    aSintDummy22 : ARRAY[0..3] OF SINT := [-128, 127, -34, 104];
    bSintDummy22 : ARRAY[0..3] OF SINT := [-128, 127, -34, 105];

    aSintDummy23 : ARRAY[0..3] OF SINT := [-128, 127, -34, 106];
    bSintDummy23 : ARRAY[0..3] OF SINT := [-128, 127, -34, 107];

    aSintDummy24 : ARRAY[0..3] OF SINT := [-128, 127, -34, 108];
    bSintDummy24 : ARRAY[0..3] OF SINT := [-128, 127, -34, 109];

    aSintDummy25 : ARRAY[0..3] OF SINT := [-128, 127, -34, 110];
    bSintDummy25 : ARRAY[0..3] OF SINT := [-128, 127, -34, 111];

    aSintDummy26 : ARRAY[0..3] OF SINT := [-128, 127, -34, 112];
    bSintDummy26 : ARRAY[0..3] OF SINT := [-128, 127, -34, 113];
END_VAR
TEST('TestWith46FailedArrayAssertions');

AssertArrayEquals_BOOL(Expecteds := aBool,
                       Actuals := bBool,
                       Message := 'Arrays differ');

AssertArrayEquals_BYTE(Expecteds := aByte,
                       Actuals := bByte,
                       Message := 'Arrays differ');

AssertArrayEquals_DINT(Expecteds := aDint,
                       Actuals := bDint,
                       Message := 'Arrays differ');

AssertArrayEquals_DWORD(Expecteds := aDword,
                        Actuals := bDword,
                        Message := 'Arrays differ');

AssertArrayEquals_DWORD(Expecteds := aDword2,
                        Actuals := bDword2,
                        Message := 'Arrays differ');

AssertArrayEquals_INT(Expecteds := aInt,
                      Actuals := bInt,
                      Message := 'Arrays differ');

AssertArrayEquals_LINT(Expecteds := aLint,
                      Actuals := bLint,
                      Message := 'Arrays differ');

AssertArrayEquals_LREAL(Expecteds := aLreal,
                        Actuals := bLreal,
                        Delta := 0.01,
                        Message := 'Arrays differ');

AssertArray2dEquals_LREAL(Expecteds := aLreal2d,
                          Actuals := bLreal2d,
                          Delta := 0.01,
                          Message := 'Arrays differ');

AssertArray3dEquals_LREAL(Expecteds := aLreal3d,
                          Actuals := bLreal3d,
                          Delta := 0.01,
                          Message := 'Arrays differ');

AssertArrayEquals_LWORD(Expecteds := aLword,
                        Actuals := bLword,
                        Message := 'Arrays differ');

AssertArrayEquals_REAL(Expecteds := aReal,
                       Actuals := bReal,
                       Delta := 0.01,
                       Message := 'Arrays differ');

AssertArray2dEquals_REAL(Expecteds := aReal2d,
                         Actuals := bReal2d,
                         Delta := 0.01,
                         Message := 'Arrays differ');

AssertArray3dEquals_REAL(Expecteds := aReal3d,
                         Actuals := bReal3d,
                         Delta := 0.01,
                         Message := 'Arrays differ');

AssertArrayEquals_SINT(Expecteds := aSint,
                       Actuals := bSint,
                       Message := 'Arrays differ');

AssertArrayEquals_UDINT(Expecteds := aUdint,
                        Actuals := bUdint,
                        Message := 'Arrays differ');

AssertArrayEquals_UINT(Expecteds := aUint,
                       Actuals := bUint,
                       Message := 'Arrays differ');

AssertArrayEquals_ULINT(Expecteds := aUlint,
                        Actuals := bUlint,
                        Message := 'Arrays differ');

AssertArrayEquals_USINT(Expecteds := aUsint,
                        Actuals := bUsint,
                        Message := 'Arrays differ');

AssertArrayEquals_WORD(Expecteds := aWord,
                       Actuals := bWord,
                       Message := 'Arrays differ');

AssertArrayEquals_SINT(Expecteds := aSintDummy1,
                       Actuals := bSintDummy1,
                       Message := 'Arrays differ');

AssertArrayEquals_SINT(Expecteds := aSintDummy2,
                       Actuals := bSintDummy2,
                       Message := 'Arrays differ');

AssertArrayEquals_SINT(Expecteds := aSintDummy3,
                       Actuals := bSintDummy3,
                       Message := 'Arrays differ');

AssertArrayEquals_SINT(Expecteds := aSintDummy4,
                       Actuals := bSintDummy4,
                       Message := 'Arrays differ');

AssertArrayEquals_SINT(Expecteds := aSintDummy5,
                       Actuals := bSintDummy5,
                       Message := 'Arrays differ');

AssertArrayEquals_SINT(Expecteds := aSintDummy6,
                       Actuals := bSintDummy6,
                       Message := 'Arrays differ');

AssertArrayEquals_SINT(Expecteds := aSintDummy7,
                       Actuals := bSintDummy7,
                       Message := 'Arrays differ');

AssertArrayEquals_SINT(Expecteds := aSintDummy8,
                       Actuals := bSintDummy8,
                       Message := 'Arrays differ');

AssertArrayEquals_SINT(Expecteds := aSintDummy9,
                       Actuals := bSintDummy9,
                       Message := 'Arrays differ');

AssertArrayEquals_SINT(Expecteds := aSintDummy10,
                       Actuals := bSintDummy10,
                       Message := 'Arrays differ');

AssertArrayEquals_SINT(Expecteds := aSintDummy11,
                       Actuals := bSintDummy11,
                       Message := 'Arrays differ');

AssertArrayEquals_SINT(Expecteds := aSintDummy12,
                       Actuals := bSintDummy12,
                       Message := 'Arrays differ');

AssertArrayEquals_SINT(Expecteds := aSintDummy13,
                       Actuals := bSintDummy13,
                       Message := 'Arrays differ');

AssertArrayEquals_SINT(Expecteds := aSintDummy14,
                       Actuals := bSintDummy14,
                       Message := 'Arrays differ');

AssertArrayEquals_SINT(Expecteds := aSintDummy15,
                       Actuals := bSintDummy15,
                       Message := 'Arrays differ');

AssertArrayEquals_SINT(Expecteds := aSintDummy16,
                       Actuals := bSintDummy16,
                       Message := 'Arrays differ');

AssertArrayEquals_SINT(Expecteds := aSintDummy17,
                       Actuals := bSintDummy17,
                       Message := 'Arrays differ');

AssertArrayEquals_SINT(Expecteds := aSintDummy18,
                       Actuals := bSintDummy18,
                       Message := 'Arrays differ');

AssertArrayEquals_SINT(Expecteds := aSintDummy19,
                       Actuals := bSintDummy19,
                       Message := 'Arrays differ');

AssertArrayEquals_SINT(Expecteds := aSintDummy20,
                       Actuals := bSintDummy20,
                       Message := 'Arrays differ');

AssertArrayEquals_SINT(Expecteds := aSintDummy21,
                       Actuals := bSintDummy21,
                       Message := 'Arrays differ');

AssertArrayEquals_SINT(Expecteds := aSintDummy22,
                       Actuals := bSintDummy22,
                       Message := 'Arrays differ');

AssertArrayEquals_SINT(Expecteds := aSintDummy23,
                       Actuals := bSintDummy23,
                       Message := 'Arrays differ');

AssertArrayEquals_SINT(Expecteds := aSintDummy24,
                       Actuals := bSintDummy1,
                       Message := 'Arrays differ');

AssertArrayEquals_SINT(Expecteds := aSintDummy25,
                       Actuals := bSintDummy1,
                       Message := 'Arrays differ');

AssertArrayEquals_SINT(Expecteds := aSintDummy26,
                       Actuals := bSintDummy26,
                       Message := 'Arrays differ');

TEST_FINISHED();
END_METHOD

END_FUNCTION_BLOCK

// ---- Test/FB_TestDurationMeasurement.TcPOU
(* This testsuite tests that durations are calculated correctly by different types of test cases
    Tests are considered passing if the duration returned is reasonablly close to the expected value.
*)
FUNCTION_BLOCK FB_TestDurationMeasurement EXTENDS TcUnit.FB_TestSuite

TestNamedTest20msDurationMeasuredCorrectly();
TestOrderedTest30msDurationMeasuredCorrectly();
TestRegularTestDurationMeasuredCorrectly();

METHOD PRIVATE TestOrderedTest30msDurationMeasuredCorrectly
VAR_INST
    DelayTimer : TON;
    Counter : DINT;
END_VAR
IF TEST_ORDERED('TestOrderedTest30msDurationMeasuredCorrectly') THEN
    DelayTimer(IN := TRUE, PT := T#30ms);   

    IF delayTimer.Q THEN
        // Write the approximate duration through an assert message for use by the verifier
        AssertEquals_LREAL(0, 0.03, 0, 'Duration');
    
        TEST_FINISHED();
    END_IF
END_IF
END_METHOD

METHOD TestRegularTestDurationMeasuredCorrectly
VAR_INST
    TestExecuted : BOOL;
    TestStartedAt : LWORD;
    TestDuration : LREAL;
    Counter : DINT;
END_VAR
TEST('TestRegularTestDurationMeasuredCorrectly');

IF NOT TestExecuted THEN
    // Introduce a delay and store the time it takes for evaluation by the test
    // use an assert statement as the delay because it takes quite a bit of time
    // double the value to account for the second assert which will print the message
    TestStartedAt := F_GetCpuCounterAs64bit(GVL_TcUnit.GetCpuCounter);
    AssertEquals_LREAL(0, 10, 0, 'Duration for calculation'); 
    TestDuration := LWORD_TO_LREAL(F_GetCpuCounterAs64bit(GVL_TcUnit.GetCpuCounter) - TestStartedAt) * GVL_TcUnit.HundredNanosecondToSecond * 2.0;
    TestExecuted := TRUE;
END_IF

// Write the duration through an assert message for use by the verifier
AssertEquals_LREAL(0, TestDuration, 0, 'Duration');

TEST_FINISHED();
END_METHOD

METHOD TestNamedTest20msDurationMeasuredCorrectly
VAR_INST
    delayTimer : TON;
END_VAR
TEST('TestNamedTest20msDurationMeasuredCorrectly');

delayTimer(IN := TRUE, PT := T#20ms);

IF delayTimer.Q THEN       
    // Write the approximate duration through an assert message for use by the verifier
    AssertEquals_LREAL(0, 0.02, 0, 'Duration');
    
    TEST_FINISHED_NAMED('TestNamedTest20msDurationMeasuredCorrectly');
END_IF
END_METHOD

END_FUNCTION_BLOCK

// ---- Test/FB_TestFileControl.TcPOU
(*
    Contains tests that verify the FileControl function block methods
*)
FUNCTION_BLOCK FB_TestFileControl EXTENDS TcUnit.FB_TestSuite

Test_FileRead();
Test_FileOpen();
Test_FileWrite();
Test_FileClose();
Test_FileDelete();

METHOD Test_FileClose
VAR
    FileControl : TcUnit.FB_FileControl;
    TestFile : STRING := 'Test_FileClose.txt';
    Mode : SysFile.ACCESS_MODE := SysFile.ACCESS_MODE.AM_APPEND_PLUS;
    Actual : SysFile.SysTypes.RTS_IEC_RESULT;
END_VAR
TEST('Test_FileClose');

FileControl.Open(TestFile, Mode);
Actual := FileControl.Close();

AssertEquals_UDINT(Expected := SysDir.CmpErrors.Errors.ERR_OK,
                   Actual := Actual,
                   Message := 'File close failed');

FileControl.Delete(TestFile);

TEST_FINISHED();
END_METHOD

METHOD Test_FileDelete
VAR
    FileControl : TcUnit.FB_FileControl;
    TestFile : STRING := 'Test_FileDelete.txt';
    Mode : SysFile.ACCESS_MODE := SysFile.ACCESS_MODE.AM_APPEND_PLUS;
    Actual : SysFile.SysTypes.RTS_IEC_RESULT;
END_VAR
TEST('Test_FileDelete');

FileControl.Open(TestFile, Mode);
FileControl.Close();
Actual := FileControl.Delete(TestFile);

AssertEquals_UDINT(Expected := Sysdir.CmpErrors.Errors.ERR_OK,
                   Actual := Actual,
                   Message := 'File deletion failed');

TEST_FINISHED();
END_METHOD

METHOD Test_FileOpen
VAR
    FileControl : FB_FileControl;
    TestFile : STRING := 'Test_FileOpen.txt';
    Mode : SysFile.ACCESS_MODE := SysFile.ACCESS_MODE.AM_APPEND_PLUS;
    Actual : SysFile.SysTypes.RTS_IEC_RESULT;
END_VAR
TEST('Test_FileOpen');

FileControl.Open(TestFile, Mode);

AssertEquals_UDINT(Expected := Sysdir.CmpErrors.Errors.ERR_OK,
                   Actual := Actual,
                   Message := 'File open failed');

FileControl.Close();
FileControl.Delete(TestFile);

TEST_FINISHED();
END_METHOD

METHOD Test_FileRead
VAR
    FileControl : FB_FileControl;
    TestFile : STRING := 'Test_FileRead.txt';
    Mode : SysFile.ACCESS_MODE := SysFile.ACCESS_MODE.AM_APPEND_PLUS;
    Result : SysFile.SysTypes.RTS_IEC_RESULT;
    FileSize : SysFile.SysTypes.RTS_IEC_SIZE;
    WriteContents : STRING(64) := '0KflxSh6C%ixPs8ReCPwFuJu)D$p*qfi66iTj&YKMdpq*EGBGiwgAsOs1s(dci';
    ReadContents : STRING(64);
END_VAR
TEST('Test_FileRead');

FileControl.Open(TestFile, Mode);
FileControl.Write(BufferPointer := ADR(WriteContents), Size := SIZEOF(WriteContents));
FileControl.Close();
FileControl.Open(TestFile, FileAccessMode := SysFile.AM_READ);

Result := FileControl.Read(BufferPointer := ADR(ReadContents), SIZEOF(ReadContents), FileSize => FileSize);

AssertEquals_STRING(Expected := WriteContents,
                    Actual := ReadContents,
                    Message := 'File read failed');

FileControl.Close();
FileControl.Delete(TestFile);

TEST_FINISHED();
END_METHOD

METHOD Test_FileWrite
VAR
    FileControl : FB_FileControl;
    Contents : STRING(64) := 'G#NkAM%Muah+nbwAk&8MnQZ9csi*YAoiGkcKzwvsYz5k@yY)aOz&cvQxXQyI6c';
    TestFile : STRING := 'Test_FileWrite.txt';
    Mode : SysFile.ACCESS_MODE := SysFile.ACCESS_MODE.AM_APPEND_PLUS;
    Actual : SysFile.SysTypes.RTS_IEC_RESULT;
END_VAR
TEST('Test_FileWrite');

FileControl.Open(TestFile, Mode);
Actual := FileControl.Write(BufferPointer := ADR(Contents), Size := SIZEOF(Contents));

AssertEquals_UDINT(Expected := SysDir.CmpErrors.Errors.ERR_OK,
                   Actual := Actual,
                   Message := 'File write failed');

FileControl.Close();
FileControl.Delete(TestFile);

TEST_FINISHED();
END_METHOD

END_FUNCTION_BLOCK

// ---- Test/FB_TestXmlControl.TcPOU
// Contains tests that verify the XmlControl function block methods
FUNCTION_BLOCK FB_TestXmlControl EXTENDS TcUnit.FB_TestSuite
VAR
    Buffer: ARRAY[0..TcUnit.GVL_Param_TcUnit.xUnitBufferSize - 1] OF BYTE;
END_VAR

Test_NewTag();
Test_NewTagNested();
Test_NewParameter();
Test_NewComment();
Test_CloseOpenTag();
Test_CloseTag();
Test_NewTagData();

METHOD PRIVATE Setup
// Clear buffer
MEMSET(ADR(Buffer), 0, SIZEOF(Buffer));
END_METHOD

METHOD PRIVATE Test_CloseOpenTag
VAR
    XmlControl : FB_XmlControl;
    TagName : STRING := 'MyTag';
    ExpectedBuffer : STRING := '<MyTag/>';
    ActualBuffer : STRING;
    ExpectedResult : STRING;
    ActualResult : STRING;
END_VAR
TEST('Test_CloseOpenTag');

Setup();

XmlControl.SetBuffer(ADR(Buffer), SIZEOF(Buffer));
XmlControl.NewTag(TagName);
XmlControl.CloseTag();
MEMCPY(ADR(ActualBuffer), ADR(Buffer), SIZEOF(ActualBuffer));

AssertEquals_String(Expected := ExpectedBuffer,
                    Actual :=  ActualBuffer,
                    Message := 'Buffer does not contain expected content');

AssertEquals_String(Expected := ExpectedResult,
                    Actual :=  ActualResult,
                    Message := 'CloseTag result does not contain expected content');

TEST_FINISHED();
END_METHOD

METHOD PRIVATE Test_CloseTag
VAR
    XmlControl : FB_XmlControl;
    TagName : STRING := 'MyTag';
    ExpectedBuffer : STRING := '<MyTag>TagData</MyTag>';
    ActualBuffer : STRING;
    ExpectedResult : STRING := '/MyTag';
    ActualResult : STRING;
END_VAR
TEST('Test_CloseTag');

Setup();

XmlControl.SetBuffer(ADR(Buffer), SIZEOF(Buffer));
XmlControl.NewTag(TagName);
XmlControl.NewTagData('TagData');
ActualResult := XmlControl.CloseTag();
MEMCPY(ADR(ActualBuffer), ADR(Buffer), SIZEOF(ActualBuffer));

AssertEquals_String(Expected := ExpectedBuffer,
                    Actual :=  ActualBuffer,
                    Message := 'Buffer does not contain expected content');

AssertEquals_String(Expected := ExpectedResult,
                    Actual :=  ActualResult,
                    Message := 'CloseTag result does not contain expected content');
                   
TEST_FINISHED();
END_METHOD

METHOD PRIVATE Test_NewComment
VAR
    XmlControl : FB_XmlControl;
    Comment : STRING := 'MyComment';
    ExpectedBuffer : STRING := '<!-- MyComment -->';
    ActualBuffer : STRING;
END_VAR
TEST('Test_NewComment');

Setup();

XmlControl.SetBuffer(ADR(Buffer), SIZEOF(Buffer));
XmlControl.NewComment(Comment);
MEMCPY(ADR(ActualBuffer), ADR(Buffer), SIZEOF(ActualBuffer));

AssertEquals_String(Expected := ExpectedBuffer,
                    Actual :=  ActualBuffer,
                    Message := 'Buffer does not contain expected content');

TEST_FINISHED();
END_METHOD

METHOD PRIVATE Test_NewParameter
VAR
    XmlControl : FB_XmlControl;
    ParameterName : STRING := 'ParaName';
    ParameterValue : STRING := 'Value';
    ExpectedBuffer : STRING := ' ParaName="Value"';
    ActualBuffer : STRING;
END_VAR
TEST('Test_NewParameter');

Setup();

XmlControl.SetBuffer(ADR(Buffer), SIZEOF(Buffer));
XmlControl.NewParameter(ParameterName, ParameterValue);
MEMCPY(ADR(ActualBuffer), ADR(Buffer), SIZEOF(ActualBuffer));

AssertEquals_String(Expected := ExpectedBuffer,
                    Actual :=  ActualBuffer,
                    Message := 'Buffer does not contain expected content');

TEST_FINISHED();
END_METHOD

METHOD PRIVATE Test_NewTag
VAR
    XmlControl : FB_XmlControl;
    TagName : STRING := 'MyTag';
    ExpectedBuffer : STRING := '<MyTag';
    ActualBuffer : STRING;
END_VAR
TEST('Test_NewTag');

Setup();

XmlControl.SetBuffer(ADR(Buffer), SIZEOF(Buffer));
XmlControl.NewTag(TagName);
MEMCPY(ADR(ActualBuffer), ADR(Buffer), SIZEOF(ActualBuffer));

AssertEquals_String(Expected := ExpectedBuffer,
                    Actual :=  ActualBuffer,
                    Message := 'Buffer does not contain expected content');

TEST_FINISHED();
END_METHOD

METHOD PRIVATE Test_NewTagData
VAR
    XmlControl : FB_XmlControl;
    TagName : STRING := 'MyTag';
    ExpectedBuffer : STRING := '<MyTag>TagData';
    ActualBuffer : STRING;
END_VAR
TEST('Test_NewTagData');

Setup();
XmlControl.SetBuffer(ADR(Buffer), SIZEOF(Buffer));
XmlControl.NewTag(TagName);
XmlControl.NewTagData('TagData');

MEMCPY(ADR(ActualBuffer), ADR(Buffer), SIZEOF(ActualBuffer));

AssertEquals_String(Expected := ExpectedBuffer,
                    Actual :=  ActualBuffer,
                    Message := 'Buffer does not contain expected content');

TEST_FINISHED();
END_METHOD

METHOD PRIVATE Test_NewTagNested
VAR
    XmlControl : FB_XmlControl;
    Tag1Name : STRING := 'MyTag1';
    Tag2Name : STRING := 'MyTag2';
    Tag3Name : STRING := 'MyTag3';
    Tag4Name : STRING := 'MyTag4';
    ExpectedBuffer : STRING := '<MyTag1><MyTag2/><MyTag3/><MyTag4/></MyTag1>';
    ActualBuffer : STRING;
END_VAR
TEST('Test_NewTagNested');

Setup();
XmlControl.SetBuffer(ADR(Buffer), SIZEOF(Buffer));

// <MyTag1><MyTag2/><MyTag3/><MyTag4/></MyTag1>
XmlControl.NewTag(Tag1Name);
XmlControl.NewTag(Tag2Name);
XmlControl.CloseTag();
XmlControl.NewTag(Tag3Name);
XmlControl.CloseTag();
XmlControl.NewTag(Tag4Name);
XmlControl.CloseTag();
XmlControl.CloseTag();

MEMCPY(ADR(ActualBuffer), ADR(Buffer), SIZEOF(ActualBuffer));

AssertEquals_String(Expected := ExpectedBuffer,
                    Actual :=  ActualBuffer,
                    Message := 'Buffer does not contain expected content');

TEST_FINISHED();
END_METHOD

END_FUNCTION_BLOCK

// ---- Test/FB_TestStreamBuffer.TcPOU
// Contains tests that verify the StreamBuffer function block methods
FUNCTION_BLOCK FB_TestStreamBuffer EXTENDS TcUnit.FB_TestSuite
VAR
    Buffer: ARRAY [0..TcUnit.GVL_Param_TcUnit.XUnitBufferSize - 1] OF BYTE;
END_VAR

Test_BufferSize();
Test_Length();
Test_Append();
Test_Clear();
Test_Find();
Test_Copy();
Test_CutOff();
Test_BufferOverflow();

METHOD PRIVATE Setup
// Clear buffer
MEMSET(ADR(Buffer), 0, SIZEOF(Buffer));
END_METHOD

METHOD PRIVATE Test_Append
VAR
    Stream : FB_StreamBuffer;
    Str1 : STRING := 'Vita est dolor sic ars.';
    Str2 : STRING := 'Vincit qui se vincit.  ';
    Search : STRING := 'se';
    TestResult : BOOL;
END_VAR
TEST('Test_Append');

Setup();

Stream.Setbuffer(ADR(Buffer), SIZEOF(Buffer));
Stream.Append := Str1;
Stream.Append := Str2;

// Search
TestResult := (Stream.Find(SearchString := Search, StartPos := 1) >= 0);

AssertTrue(Condition := TestResult,
           Message := 'Append failed');

TEST_FINISHED();
END_METHOD

METHOD Test_BufferOverflow
VAR
    Stream : FB_StreamBuffer;
    Str1 : STRING := 'abcdef';
    Str2 : STRING := 'uwxyz';
    Cpy : STRING;
    CopyLen : UDINT;
    SmallBuffer : ARRAY [0..SMALL_BUFFER_SIZE-1] OF BYTE;
END_VAR
VAR CONSTANT
    SMALL_BUFFER_SIZE : UDINT := 10;
END_VAR
TEST('Test_BufferOverflow');

Setup();

Stream.SetBuffer(ADR(SmallBuffer), SIZEOF(SmallBuffer));
Stream.Append := Str1;
Stream.Append := Str2;

AssertEquals_UDINT(SMALL_BUFFER_SIZE, Stream.Length, 'Stream not at maximum length');

Cpy := Stream.Copy(StartPos := 1, EndPos := Stream.Length, CopyLen => CopyLen);

// Expected behavior: the buffer receives up to Buffer Size - 1 of string, the last byte is NULL character (termination)
AssertEquals_STRING(Expected := 'abcdefuwx',
                    Actual := Cpy,
                    Message := 'Stream was not truncated as expected');

TEST_FINISHED();
END_METHOD

METHOD PRIVATE Test_BufferSize
VAR
    Stream : FB_StreamBuffer;
END_VAR
TEST('Test_BufferSize');

Setup();

Stream.Setbuffer(ADR(Buffer), SIZEOF(Buffer));

// Compare initialised buffersize with expected buffersize
AssertEquals_UDINT(Expected := GVL_Param_TcUnit.xUnitBufferSize,
                   Actual := Stream.BufferSize,
                   Message := 'BufferSize differs');

TEST_FINISHED();
END_METHOD

METHOD PRIVATE Test_Clear
VAR
    Stream : FB_StreamBuffer;
    Str : STRING := 'vita est dolor sic ars';
END_VAR
TEST('Test_Clear');

Setup();

Stream.Setbuffer(ADR(Buffer), SIZEOF(Buffer));
Stream.Append := Str;
Stream.Clear();

AssertEquals_UDINT(Expected := 0,
                   Actual := Stream.Length, 
                   Message := 'Length differs');

TEST_FINISHED();
END_METHOD

METHOD PRIVATE Test_Copy
VAR
    Stream : FB_StreamBuffer;
    Str1 : STRING := 'Vincit qui se vincit.  ';
    Str2 : STRING := 'Vita est dolor sic ars.';
    Cpy : STRING;
    CopyLen : UDINT;
END_VAR
TEST('Test_Copy');

Setup();

Stream.Setbuffer(ADR(Buffer), SIZEOF(Buffer));
Stream.Append := Str1;
Stream.Append := Str2;

// Copy from 8th char 3 chars (8+3=11), should be 'qui'
Cpy := Stream.Copy(StartPos := 8, EndPos := 11, CopyLen => CopyLen);

AssertEquals_STRING(Expected := 'qui',
                    Actual := Cpy,
                    Message := 'Copy Failed');

TEST_FINISHED();
END_METHOD

METHOD PRIVATE Test_CutOff
VAR
    Stream : FB_StreamBuffer;
    Str : STRING := 'vita est dolor sic ars';
    Cut : UDINT;
    Length : UDINT;
    CutOff : STRING;
    Expected : STRING;
END_VAR
TEST('Test_CutOff');

Setup();

Stream.Setbuffer(ADR(Buffer), SIZEOF(Buffer));

// Last char - 2 chars = 3 chars in total
Stream.Append := Str;
Cut := (Stream.Length - 2); 

// CutOff should contain 'ars'
CutOff := Stream.CutOff(StartPos := Cut, CutLen => Length);
Expected := Stream.Copy(StartPos := 1, EndPos := Stream.Length); 

AssertEquals_String(Expected := Expected, 
                    Actual := 'vita est dolor sic',
                    Message := 'CutOff string differs');

TEST_FINISHED();
END_METHOD

METHOD PRIVATE Test_Find
VAR
    Stream : FB_StreamBuffer;
    Str : STRING := 'Vita est dolor sic ars.';
    Search : STRING := 'dolor';
    TestResult : BOOL;
END_VAR
TEST('Test_Find');

Setup();

Stream.Setbuffer(ADR(Buffer), SIZEOF(Buffer));
Stream.Append:= Str;

// Start search at 1st char
TestResult := (Stream.Find(SearchString := Str, StartPos := 1 ) >= 0); 

AssertTrue(Condition := TestResult,
           Message := 'Find Failed');

TEST_FINISHED();
END_METHOD

METHOD PRIVATE Test_Length
VAR
    Stream : FB_StreamBuffer;
    Str : STRING := 'vita est dolor sic ars';
    Length : UDINT;
END_VAR
TEST('Test_Length');

Setup();

Stream.Setbuffer(ADR(Buffer), SIZEOF(Buffer));
Stream.Append := Str;
Length := TO_UDINT(LEN(Str));

AssertEquals_UDINT(Expected := length,
                   Actual := Stream.Length,
                   Message := 'Length differs');

TEST_FINISHED();
END_METHOD

END_FUNCTION_BLOCK

// ---- Test/FB_TestFinishedNamed.TcPOU
(* This function blocks tests the TEST_FINISHED_NAMED function by creating various tests
   and finishing them in steps *)
FUNCTION_BLOCK FB_TestFinishedNamed EXTENDS TcUnit.FB_TestSuite
VAR
END_VAR

END_FUNCTION_BLOCK

// ---- Test/FB_EmptyAssertionMessage.TcPOU
(* This testsuite creates a failed test with an empty assertion message *)
FUNCTION_BLOCK FB_EmptyAssertionMessage EXTENDS TcUnit.FB_TestSuite

IntegerEmptyAssertionMessage();

METHOD PRIVATE IntegerEmptyAssertionMessage
VAR
    a : INT := -32000;
    b : INT := 15423;
END_VAR
TEST('IntegerEmptyAssertionMessage');

AssertEquals_INT(Expected := a,
                 Actual := b,
                 Message := '');

TEST_FINISHED();
END_METHOD

END_FUNCTION_BLOCK

// ---- Test/FB_AssertCountExceedsMaxNumber.TcPOU
(*
    This test-suite runs several asserts with the same parameters (same expected, actual, message), calling the asserts
    in different cycles and using the same test.
    On top of this, we will call new asserts (though with same parameters) in later cycles.
    The reason we want the framework to support this is that theoretically the user could want to do an assert with the
    same message, using the same test with the same data values for both expected and actual, and splitting the asserts
    on different cycles.
*)
FUNCTION_BLOCK FB_AssertCountExceedsMaxNumber EXTENDS TcUnit.FB_TestSuite
VAR
END_VAR

Assert_SameEntryInOneCycle();
Assert_SameArrayEntryInOneCycle();

METHOD PRIVATE Assert_SameArrayEntryInOneCycle
VAR
    a : ARRAY[1..ARRAY_LENGTH] OF DWORD := [16#12345678, 16#23456789];
    b : ARRAY[1..ARRAY_LENGTH] OF DWORD := [16#90ABCDEF, 16#0ABCDEF1];

	i : UINT;
END_VAR
VAR CONSTANT
	ARRAY_LENGTH : UINT := 2;
	MAX_INDEX : UINT := (TcUnit.GVL_Param_TcUnit.MaxNumberOfAssertsForEachTestSuite + 100);
END_VAR
TEST('Assert_SameArrayEntryInOneCycle');

// Only checks if PLC crashes
FOR i := 1 TO MAX_INDEX DO
	AssertArrayEquals_DWORD(Expecteds := a,
						   	Actuals := a,
						   	Message := 'Values differ');
END_FOR;

AssertEquals_UINT(Expected := GVL_Param_TcUnit.MaxNumberOfAssertsForEachTestSuite,
		          Actual := AssertArrayResults.TotalArrayAsserts,
		          Message := 'AssertArrayResults.TotalArrayAsserts invalid');

TEST_FINISHED();
END_METHOD

METHOD PRIVATE Assert_SameEntryInOneCycle
VAR
    a : DWORD := 16#12345678;
    b : DWORD := 16#90ABCDEF;

	i : UINT;
END_VAR
VAR CONSTANT
	MAX_INDEX : UINT := (TcUnit.GVL_Param_TcUnit.MaxNumberOfAssertsForEachTestSuite + 100); 
END_VAR
TEST('Assert_SameEntryInOneCycle');

// Only checks if PLC crashes
FOR i := 1 TO MAX_INDEX DO
	AssertEquals_DWORD(Expected := a,
					   Actual := a,
					   Message := 'Values differ');
END_FOR;

AssertEquals_UINT(Expected := GVL_Param_TcUnit.MaxNumberOfAssertsForEachTestSuite,
		          Actual := AssertResults.TotalAsserts,
		          Message := 'AssertResults.TotalAsserts invalid');

TEST_FINISHED();
END_METHOD

END_FUNCTION_BLOCK

// ---- Test/FB_TestFinishedNamedDoesNotExist.TcPOU
(*
    This FB tests the free function TEST_FINISHED_NAMED. Calling this function with a name that doesn't exist should
    produce an error message that says so. This error message should also only be printed once.
*)
FUNCTION_BLOCK FB_TestFinishedNamedDoesNotExist EXTENDS TcUnit.FB_TestSuite
VAR
END_VAR

Test_FinishedNamed();

METHOD PRIVATE Test_FinishedNamed
VAR
    a : INT := 2;
    b : INT := 2;
END_VAR
TEST('Test_FinishedNamed');

AssertEquals_INT(Expected := a,
                 Actual := b,
                 Message := 'Values differ');

TEST_FINISHED_NAMED('AnotherTestNameThatDoesNotExist');
END_METHOD

END_FUNCTION_BLOCK
